{attribute 'qualified_only'}
VAR_GLOBAL CONSTANT
	analogOutputMaxVolt : INT := 10;
	intMaxValue : INT :=32767;
	samplingTime : REAL := 1000;
	globAnalogOutput AT %Q* : INT;
END_VAR

(* stored: Version 1.1.0.1, ProductVersion 3.1.4022.12
   GVL GVL_1: Id {7aa005aa-e593-4977-b375-8931f5877994} *)
